(*====================================
				下壓放
  ====================================*) 
		
	9340:
		GroupFx.A_UnPress();
		GroupFx.C_UnPress();
		step := step + 1;
		
	9341:
		IF (GroupFx.step_A_P.bBuzy OR GroupFx.step_A_P.bError) AND
			(GroupFx.step_C_P.bBuzy OR GroupFx.step_C_P.bError) THEN
			step := step + 1;
		END_IF
		
	9342:
		IF (GroupFx.step_A_P.bDone AND GroupFx.step_A_P.bDone) OR
			GroupFx.step_C_P.bError OR GroupFx.step_C_P.bError OR
			NOT Hmi_Web.Jog_FxA.V_Open THEN
			step := 9349;
		END_IF
		
	9349:
		IF NOT Hmi_Web.Jog_FxA.V_Open THEN
			step:=8001;
		END_IF
		
(*====================================
				滾輪正轉
  ====================================*) 
		
	9360:
		Fx.RelMove(100000, 200 * Hmi.Jog_Speed * 0.01);
		step := step + 1;
		
	9361:
		IF Fx.bDone OR Fx.bError OR NOT Hmi_Web.Jog_FxA.P THEN
			step := 9369;
		END_IF
		
	9369:
		Fx.Stop();
		IF NOT Hmi_Web.Jog_FxA.P THEN
			step:=8001;
		END_IF
(*====================================
				滾輪反轉
  ====================================*) 
		
	9370:
		Fx.RelMove(-100000, 200 * Hmi.Jog_Speed * 0.01);
		step := step + 1;
		
	9371:
		IF Fx.bDone OR Fx.bError OR NOT Hmi_Web.Jog_FxA.N THEN
			step := 9389;
		END_IF
		
	9379:
		Fx.Stop();
		IF NOT Hmi_Web.Jog_FxA.N THEN
			step:=8001;
		END_IF
		
END_CASE
END_ACTION

ACTION step_9400_Jog_GroupFx_B:
(*====================================
		Group FX B軸 Jog模式
  ====================================*) 

CASE step OF
(*	====================================
					夾
  ====================================*) 

	9400: // 夾
		IF NOT io.i502 AND NOT io.i504 THEN
			GroupFx.BD_Clamp();
			step := step + 1;
		ELSE
			IF NOT io.i502 THEN
				pMsg.Push_alarm("JOG FxB: B下壓不再原點上");
			END_IF
			IF NOT io.i504 THEN
				pMsg.Push_alarm("JOG FxB: D下壓不再原點上");
			END_IF
			step := 9409;
		END_IF
		
		
	9401:
		IF GroupFx.step_BD_C.bBuzy OR NOT Hmi_Web.Jog_FxB.H_Close THEN
			step := step + 1;
		END_IF
		
	9402:
		IF GroupFx.step_BD_C.bDone OR NOT Hmi_Web.Jog_FxB.H_Close THEN
			step:=9409;
		END_IF
		
	9409:
		GroupFx.BD_Stop();
		IF NOT Hmi_Web.Jog_FxB.H_Close THEN
			step:=8001;
		END_IF

(*	====================================
					保持
	====================================	*) 
	9410:
		IF GroupFx.b_BD_Clamp THEN
			GroupFx.BD_Clamp();
			step := step + 1;
		ELSE
			step := 9419;
			pMsg.Push_alarm("JOG FxB: 尚未執行FxB夾輪靠緊");
		END_IF
		
	9411:
		IF GroupFx.step_BD_C.bBuzy OR GroupFx.step_BD_C.bError THEN
			step := step + 1;
		END_IF
		
	9412:
		IF GroupFx.step_BD_C.bdone THEN
			step := step + 1;
		ELSIF GroupFx.step_BD_C.bError THEN
			pMsg.Push_alarm("JOG FxB: 執行FxB夾輪保持時發生錯誤");
		END_IF
		
	9413:
		Hmi_Web.Jog_FxB.H_Hold := FALSE;
		step:=9419;
		
	9419:
		step:=8001;

(*	====================================
					放
  	====================================*) 
	9420: // 放
		IF NOT io.i502 AND NOT io.i504 THEN
			GroupFx.BD_UnClamp(99999);
			step := step + 1;
		ELSE
			IF io.i502 THEN
				pMsg.Push_alarm("JOG FxB: B下壓不再原點上");
			END_IF
			IF io.i504 THEN
				pMsg.Push_alarm("JOG FxB: D下壓不再原點上");
			END_IF
			step := 9429;
		END_IF
		
	9421:
		IF GroupFx.step_BD_C.bBuzy OR NOT Hmi_Web.Jog_FxB.H_Open THEN
			step := step + 1;
		END_IF
		
	9422:
		IF GroupFx.step_BD_C.bDone OR NOT Hmi_Web.Jog_FxB.H_Open THEN
				step:=9429;
		END_IF
		
	9429:
		GroupFx.BD_Stop();
		IF NOT Hmi_Web.Jog_FxB.H_Open THEN
			step:=8001;
		END_IF
		
(*	====================================
					下壓夾
  	====================================*) 
		
	9430:
		GroupFx.B_Press();
		GroupFx.D_Press();
		step := step + 1;
		
	9431:
		IF (GroupFx.step_B_P.bBuzy OR GroupFx.step_B_P.bError) AND
			(GroupFx.step_D_P.bBuzy OR GroupFx.step_D_P.bError) THEN
			step := step + 1;
		END_IF
		
	9432:
		IF (GroupFx.step_B_P.bDone AND GroupFx.step_B_P.bDone) OR
			GroupFx.step_D_P.bError OR GroupFx.step_D_P.bError OR
			NOT Hmi_Web.Jog_FxB.V_Close THEN
			step := 9439;
		END_IF
		
	9439:
		IF NOT Hmi_Web.Jog_FxB.V_Close THEN
			step:=8001;
		END_IF
		
(*	====================================
					下壓放
  	====================================*) 
		
	9440:
		GroupFx.B_UnPress();
		GroupFx.D_UnPress();
		step := step + 1;
		
	9441:
		IF (GroupFx.step_B_P.bBuzy OR GroupFx.step_B_P.bError) AND
			(GroupFx.step_D_P.bBuzy OR GroupFx.step_D_P.bError) THEN
			step := step + 1;
		END_IF
		
	9442:
		IF (GroupFx.step_B_P.bDone AND GroupFx.step_B_P.bDone) OR
			GroupFx.step_D_P.bError OR GroupFx.step_D_P.bError OR
			NOT Hmi_Web.Jog_FxB.V_Open THEN
			step := 9449;
		END_IF
		
	9449:
		IF NOT Hmi_Web.Jog_FxB.V_Open THEN
			step:=8001;
		END_IF
END_CASE
END_ACTION

ACTION step_9700_Jog_SetLimit:
(*====================================
				設定極限
  ====================================*) 

CASE step OF
	9700:
		IF Hmi.Jog_GroupSelect > 0 THEN
			IF Hmi.Set_X_P_Limite THEN
				step := 9710;
			ELSIF Hmi.Set_X_Home THEN
				step := 9720;
			ELSIF Hmi.Set_Y_P_Limite THEN
				step := 9730;
			ELSIF Hmi.Set_Y_Home THEN
				step := 9740;
			ELSIF Hmi.Set_Z_P_Limite THEN
				step := 9750;
			ELSIF Hmi.Set_Z_Home THEN
				step := 9760;
			ELSE
				step := step + 1;
			END_IF
		ELSE
			Hmi.Set_X_P_Limite := FALSE;
			Hmi.Set_X_Home := FALSE;
			Hmi.Set_Y_P_Limite := FALSE;
			Hmi.Set_Y_Home := FALSE;
			Hmi.Set_Z_P_Limite := FALSE;
			Hmi.Set_Z_Home := FALSE;
			step := step + 1;
		END_IF
		
	9701:
		IF Hmi.Mode_Select = 1 THEN
			step := 8000;
		ELSIF Hmi.Mode_Select = 2 THEN
			step := 8010;
		ELSE
			step := 0;
		END_IF
		


(*====================================
				X+
  ====================================*)
	9710:
		CASE Hmi.Jog_GroupSelect OF
			1:
				posc.GaX_P_Limite := GaX.Pos + 2;
				GaX.SetLimit();
				step := step + 1;
				
			2:
				posc.GbX_P_Limite := GbX.Pos + 2;
				GbX.SetLimit();
				step := step + 1;
				
			3:
				posc.GcX_P_Limite := GcX.Pos + 2;
				GcX.SetLimit();
				step := step + 1;
				
			4:
				posc.GdX_P_Limite := GdX.Pos + 2;
				GdX.SetLimit();
				step := step + 1;
				
			ELSE
				step := 9700;
		END_CASE
		
		
	9711:
		Hmi.Set_X_P_Limite := FALSE;
		step := 9790;
		
(*====================================
				X-
  ====================================*) 
  	9720:
		CASE Hmi.Jog_GroupSelect OF
			1:
				posc.GaX_N_Limite := -2;
				GaX.Homing();
				step := step + 1;
				
			2:
				posc.GbX_N_Limite := -2;
				GbX.Homing();
				step := step + 1;
				
			3:
				posc.GcX_N_Limite := -2;
				GcX.Homing();
				step := step + 1;
				
			4:
				posc.GdX_N_Limite := -2;
				GdX.Homing();
				step := step + 1;
				
			ELSE
				step := 9700;
		END_CASE
		
		
	9721:
		IF (Hmi.Jog_GroupSelect = 1 AND (GaX.bBuzy OR GaX.bError)) OR 
			(Hmi.Jog_GroupSelect = 2 AND (GbX.bBuzy OR GbX.bError)) OR
			(Hmi.Jog_GroupSelect = 3 AND (GcX.bBuzy OR GcX.bError)) OR
			(Hmi.Jog_GroupSelect = 4 AND (GdX.bBuzy OR GdX.bError)) 
		THEN
			step := step + 1;
		END_IF
		
	9722:
		IF (Hmi.Jog_GroupSelect = 1 AND GaX.bDone) OR
			(Hmi.Jog_GroupSelect = 1 AND GbX.bDone) OR
			(Hmi.Jog_GroupSelect = 3 AND GcX.bDone) OR
			(Hmi.Jog_GroupSelect = 4 AND GdX.bDone)
		THEN
			step := step + 1;
		ELSIF (Hmi.Jog_GroupSelect = 1 AND GaX.bError) OR
			(Hmi.Jog_GroupSelect = 1 AND GbX.bError) OR
			(Hmi.Jog_GroupSelect = 3 AND GcX.bError) OR
			(Hmi.Jog_GroupSelect = 4 AND GdX.bError)
		THEN
			step := 9700;
		END_IF
		
	9723:
		CASE Hmi.Jog_GroupSelect OF
			1:
				GaX.SetLimit();
				step := step + 1;
				
			2:
				GbX.SetLimit();
				step := step + 1;
				
			3:
				GcX.SetLimit();
				step := step + 1;
				
			4:
				GdX.SetLimit();
				step := step + 1;
				
			ELSE
				step := step + 1;
		END_CASE
		
	9724:	
		Hmi.Set_X_Home := FALSE;
		step := 9790;
		
(*====================================
				Y+
  ====================================*)
	9730:
		CASE Hmi.Jog_GroupSelect OF
			1:
				posc.GaY_P_Limite := GaY.Pos + 2;
				GaY.SetLimit();
				step := step + 1;
				
			2:
				posc.GbY_P_Limite := GbY.Pos + 2;
				GbY.SetLimit();
				step := step + 1;
				
			3:
				posc.GcY_P_Limite := GcY.Pos + 2;
				GcY.SetLimit();
				step := step + 1;
				
			4:
				posc.GdY_P_Limite := GdY.Pos + 2;
				GdY.SetLimit();
				step := step + 1;
				
			ELSE
				step := step + 1;
		END_CASE
		
		
	9731:
		Hmi.Set_Y_P_Limite := FALSE;
		step := 9790;
		
(*====================================
				Y-
  ====================================*) 
  	9740:
		CASE Hmi.Jog_GroupSelect OF
			1:
				posc.GaY_N_Limite := -2;
				GaY.Homing();
				step := step + 1;
				
			2:
				posc.GbY_N_Limite := -2;
				GbY.Homing();
				step := step + 1;
				
			3:
				posc.GcY_N_Limite := -2;
				GcY.Homing();
				step := step + 1;
				
			4:
				posc.GdY_N_Limite := -2;
				GdY.Homing();
				step := step + 1;
				
			ELSE
				step := 9700;
		END_CASE
		
		
	9741:
		IF (Hmi.Jog_GroupSelect = 1 AND (GaY.bBuzy OR GaY.bError)) OR 
			(Hmi.Jog_GroupSelect = 2 AND (GbY.bBuzy OR GbY.bError)) OR
			(Hmi.Jog_GroupSelect = 3 AND (GcY.bBuzy OR GcY.bError)) OR
			(Hmi.Jog_GroupSelect = 4 AND (GdY.bBuzy OR GdY.bError)) 
		THEN
			step := step + 1;
		END_IF
		
	9742:
		IF (Hmi.Jog_GroupSelect = 1 AND GaY.bDone) OR
			(Hmi.Jog_GroupSelect = 2 AND GbY.bDone) OR
			(Hmi.Jog_GroupSelect = 3 AND GcY.bDone) OR
			(Hmi.Jog_GroupSelect = 4 AND GdY.bDone)
		THEN
			step := step + 1;
		ELSIF (Hmi.Jog_GroupSelect = 1 AND GaY.bError) OR
			(Hmi.Jog_GroupSelect = 2 AND GbY.bError) OR
			(Hmi.Jog_GroupSelect = 3 AND GcY.bError) OR
			(Hmi.Jog_GroupSelect = 4 AND GdY.bError)
		THEN
			step := 9700;
		END_IF
		
	9743:
		CASE Hmi.Jog_GroupSelect OF
			1:
				GaY.SetLimit();
				step := step + 1;
				
			2:
				GbY.SetLimit();
				step := step + 1;
				
			3:
				GcY.SetLimit();
				step := step + 1;
				
			4:
				GdY.SetLimit();
				step := step + 1;
				
			ELSE
				step := step + 1;
		END_CASE
		
	9744:
		Hmi.Set_Y_Home := FALSE;
		step := 9790;
		
(*====================================
				Z+
  ====================================*)
	9750:
		CASE Hmi.Jog_GroupSelect OF
			1:
				posc.GaZ_P_Limite := GaZ.Pos + 2;
				GaZ.SetLimit();
				step := step + 1;
				
			2:
				posc.GbZ_P_Limite := GbZ.Pos + 2;
				GbZ.SetLimit();
				step := step + 1;
				
			3:
				posc.GcZ_P_Limite := GcZ.Pos + 2;
				GcZ.SetLimit();
				step := step + 1;
				
			4:
				posc.GdZ_P_Limite := GdZ.Pos + 2;
				GdZ.SetLimit();
				step := step + 1;
				
			ELSE
				step := step + 1;
		END_CASE
		
		
	9751:
		Hmi.Set_Z_P_Limite := FALSE;
		step := 9790;
		
(*====================================
				Z-
  ====================================*) 
	9760:
		CASE Hmi.Jog_GroupSelect OF
			1:
				posc.GaZ_N_Limite := -2;
				GaZ.Homing();
				step := step + 1;
				
			2:
				posc.GbZ_N_Limite := -2;
				GbZ.Homing();
				step := step + 1;
				
			3:
				posc.GcZ_N_Limite := -2;
				GcZ.Homing();
				step := step + 1;
				
			4:
				posc.GdZ_N_Limite := -2;
				GdZ.Homing();
				step := step + 1;
				
			ELSE
				step := 9700;
		END_CASE
		
		
	9761:
		IF (Hmi.Jog_GroupSelect = 1 AND (GaZ.bBuzy OR GaZ.bError)) OR 
			(Hmi.Jog_GroupSelect = 2 AND (GbZ.bBuzy OR GbZ.bError)) OR
			(Hmi.Jog_GroupSelect = 3 AND (GcZ.bBuzy OR GcZ.bError)) OR
			(Hmi.Jog_GroupSelect = 4 AND (GdZ.bBuzy OR GdZ.bError)) 
		THEN
			step := step + 1;
		END_IF
		
	9762:
		IF (Hmi.Jog_GroupSelect = 1 AND GaZ.bDone) OR
			(Hmi.Jog_GroupSelect = 1 AND GbZ.bDone) OR
			(Hmi.Jog_GroupSelect = 3 AND GcZ.bDone) OR
			(Hmi.Jog_GroupSelect = 4 AND GdZ.bDone)
		THEN
			step := step + 1;
		ELSIF (Hmi.Jog_GroupSelect = 1 AND GaZ.bError) OR
			(Hmi.Jog_GroupSelect = 1 AND GbZ.bError) OR
			(Hmi.Jog_GroupSelect = 3 AND GcZ.bError) OR
			(Hmi.Jog_GroupSelect = 4 AND GdZ.bError)
		THEN
			step := 9700;
		END_IF
		
	9763:
		CASE Hmi.Jog_GroupSelect OF
			1:
				GaZ.SetLimit();
				step := step + 1;
				
			2:
				GbZ.SetLimit();
				step := step + 1;
				
			3:
				GcZ.SetLimit();
				step := step + 1;
				
			4:
				GdZ.SetLimit();
				step := step + 1;
				
			ELSE
				step := step + 1;
		END_CASE
		step := step + 1;
		
	9764:
		Hmi.Set_Z_Home := FALSE;
		step := 9790;
		
		
		
	9790:
		fbWritePersistentData.START := TRUE;
		step := step  + 1;
		
	9791:
		IF NOT fbWritePersistentData.BUSY THEN
			fbWritePersistentData.START := FALSE;
			step := step  + 1;
		END_IF
		
	9792:
		step := 9700;

END_CASE
END_ACTION

ACTION Timer:
tmr01();
END_ACTION

ACTION WritePersistentData:
fbWritePersistentData(
	PORT:= 851,
	TMOUT:= T#5S, 
	MODE:= SPDM_2PASS, 
	);
END_ACTION

END_PROGRAM

(* stored: Version 1.1.0.1, ProductVersion 3.1.4026.13
   POU AutoMain: Id {640ea801-bc75-4e57-87c7-5cbed9d57d57}, SpecialFunc None
   Folder JOG流程8100_9400: Id {29c869f8-9e55-4891-96de-3fdfd31f73ae}
   Folder 內部啟動用: Id {e54b00b0-37e1-43e2-ac19-0768ee77541d}
   Folder 自動流程500_1000: Id {ed3b663e-b781-4d3b-9e19-bc41e1e6cd65}
   Folder 測試用區域: Id {91315759-1bb3-4063-b768-24ddab7b0df1}
   Folder 輔助流程_加工動作中自動進料: Id {60021586-c26a-4340-8fba-12b4e808dba8}
   Method Homming: Id {44f06067-4083-4ca2-8078-ae6d4fcf2533}
   Method JogMode: Id {762caa98-70af-49ec-be7a-f088d4acd762}
   Method JogMode_Exit: Id {5ff6d66b-3b76-4114-a060-32c154db4adc}
   Method ReStart: Id {36176bad-7a12-42cc-9d4b-bc1b6cb32850}
   Action Start_Feed_In_NC_Start: Id {b2d72d96-9689-4363-85ee-014fef8de968}
   Action Step_0_Main: Id {b79c11b6-0e6f-4d9a-8471-e672afa2103e}
   Action step_0100_Homming: Id {a8c1ccf9-ccda-4182-a22a-bf89b00c7b8b}
   Action step_0500_AutoMode_StartCheck: Id {4829e2e7-827c-4026-a87b-a346e004fcb7}
   Action step_0600_AutoMode_Feed: Id {d813016f-ba23-4674-893e-521536c59444}
   Action step_0700_AutoMode_GoPrintPoint: Id {3ddf49fc-b8c3-43b2-aa40-0220e552ab46}
   Action step_0800_AutoMode_GoPrintPoint_Cycle_200_UP: Id {b9ee8044-d68a-43ca-8ce0-75cc1609900c}
   Action step_0900_AutoMode_GoPrintPoint_Cycle_200_Down: Id {93b20725-0dc6-4893-8408-c5a0e7cf97fe}
   Action step_1000_AutoPrgEnd: Id {d4a54de3-d318-4b44-9a1a-75a485fce4e2}
   Action step_7000_test_mask_A: Id {9c11a767-a79b-4d55-b953-b21e0bc4b4a0}
   Action step_7100_test_mask_A_1: Id {5fd6c699-8423-4243-9463-d08b5464c75f}
   Action step_7200_test_mask_B: Id {4c61de62-fb3a-448e-87a0-699fa1e97c12}
   Action step_7300_test_mask_B_1: Id {8d03264d-5885-47fe-a0e0-a32c6f133f5b}
   Action step_7400_test_mask_C: Id {fc0c6fda-73e2-41af-9fc9-5032d411c6d4}
   Action step_7500_test_mask_C_1: Id {157bc15f-5e02-418c-931b-18c000d4256a}
   Action step_7600_test_mask_D: Id {0b9c3ef3-9254-45dc-bc49-5cb485e2f771}
   Action step_7700_test_mask_D_1: Id {ed775e26-4708-4de8-8dbb-4ec7681b81d3}
   Action step_7800_FindZ: Id {78554766-b253-4c2b-86e4-fe4f195d427b}
   Action step_7900_SensorTest: Id {2a2185c3-79fd-40b1-a47d-319d15089cdf}
   Action step_8000_Jog: Id {c27e7acc-5ac3-4b59-9fa3-c17028cc9d68}
   Action step_8100_Jog_GroupA_X: Id {e799dead-5ecb-44cb-96a8-211ac7ea9e16}
   Action step_8200_Jog_GroupA_Y: Id {37ce9b29-c425-42de-8468-6415230b3534}
   Action step_8300_Jog_GroupA_Z: Id {5a63ed6b-fb7d-4cb7-81bb-e4a40e19dcb5}
   Action step_8400_Jog_GroupB_X: Id {f02d0236-6e7f-4e25-a06a-ca2355ca4b9a}
   Action step_8500_Jog_GroupB_Y: Id {d9913704-7786-46a8-84b1-7db0eaf1f3b6}
   Action step_8600_Jog_GroupB_Z: Id {3c8cdb25-5cb1-4b0f-b934-e73736a2fa67}
   Action step_8700_Jog_GroupC_X: Id {7ad358ea-2217-42cd-9261-5e2d16620efe}
   Action step_8800_Jog_GroupC_Y: Id {6d571eda-dd32-4acd-9da1-545affc0a066}
   Action step_8900_Jog_GroupC_Z: Id {53227d1d-026f-48c0-ad4b-19eb9bfd66e5}
   Action step_9000_Jog_GroupD_X: Id {5db77154-6d99-4cea-89d3-6cfd264fd84d}
   Action step_9100_Jog_GroupD_Y: Id {91ffc927-82c0-469b-8f33-9a13afeabebf}
   Action step_9200_Jog_GroupD_Z: Id {2c5f3bd0-6f4a-4e8d-9ccd-8e124117a518}
   Action step_9300_Jog_GroupFx_A: Id {4ea608c7-d2b7-4028-abc8-0bf6443d9578}
   Action step_9400_Jog_GroupFx_B: Id {b3bfee0c-2d0d-4c88-a8a1-984085440ece}
   Action step_9700_Jog_SetLimit: Id {b2fe7821-cf3c-4702-8677-8a39e991af14}
   Action Timer: Id {c4f557db-fcde-4848-b204-06307f28f9ff}
   Action WritePersistentData: Id {19164537-7422-43c1-bcc7-02dc2b29a4be} *)
